{attribute 'c++_compatible'}
FUNCTION_BLOCK UDPConnect IMPLEMENTS ITcIoUdpProtocolRecv
VAR_INPUT
END_VAR
VAR_OUTPUT
END_VAR
VAR
	{attribute 'TcInitSymbol'}
    oid:              OTCID; 
    ipUdp:            ITcIoUdpProtocol;
    updPort:          UINT := 25000;
    nReceivedPakets:  UINT;
    hrInit :          HRESULT;
    hrSend :          HRESULT;
END_VAR

IF ipUdp <> 0 THEN
    ipUdp.CheckReceived();
END_IF

METHOD FB_exit : BOOL
VAR_INPUT
	bInCopyCode : BOOL; // if TRUE, the exit method is called for exiting an instance that is copied afterwards (online change).
END_VAR
IF (NOT bInCopyCode AND ipUdp <> 0) THEN //Shutdown
     ipUdp.UnregisterReceiver(updPort);
    FW_SafeRelease(ADR(ipUdp));
     FB_exit := TRUE;
ELSE
     FB_exit := FALSE;
END_IF
END_METHOD

METHOD FB_init : BOOL
VAR_INPUT
	bInitRetains : BOOL; // if TRUE, the retain variables are initialized (warm start / cold start)
	bInCopyCode : BOOL;  // if TRUE, the instance afterwards gets moved into the copy code (online change)
END_VAR

VAR
    ipSrv: ITComObjectServer;
    hr : HRESULT;
END_VAR
IF NOT bInCopyCode THEN // no online change
    IF ipUdp = 0 THEN
     hrInit := FW_ObjMgr_GetObjectInstance(   oid:=oid, 
    
    iid:=TC_GLOBAL_IID_LIST.IID_ITcIoUdpProtocol, 

    pipUnk:=ADR(ipUdp) );
        IF ( SUCCEEDED(hr) AND ipUdp.RegisterReceiver(updPort, THIS^) = 0 ) THEN //open port
            FB_init := TRUE;
        ELSE
            FB_init := FALSE; 
            FW_SafeRelease(ADR(ipUdp));
        END_IF
    END_IF
END_IF
END_METHOD

METHOD FB_reinit : BOOL
VAR_INPUT
END_VAR
IF (ipUdp <> 0) THEN 
 ipUdp.RegisterReceiver(updPort, THIS^);
END_IF
END_METHOD

{attribute 'object_name' := 'ReceiveData'}
{attribute 'c++_compatible'}
{attribute 'signature_flag' := '33554688'}
{attribute 'pack_mode' := '4'}
{attribute 'show'}
{attribute 'minimal_input_size' := '4'}
METHOD ReceiveData : HRESULT
VAR_INPUT
	ipAddr	: UDINT;
	udpDestPort	: UINT;
	udpSrcPort	: UINT;
	nData	: UDINT;
	pData	: PVOID;
	pVlan	: POINTER TO ETYPE_VLAN_HEADER := 0;
END_VAR

VAR
	i	: ULINT := 0;
END_VAR
nReceivedPakets := nReceivedPakets+1;
//MAIN_UDP.nPaketlaenge := nData;

FOR i := 0 TO 3 DO
	memcpy(ADR(UDP.x[i+1]),pData+((i*3)*8),8);
	memcpy(ADR(UDP.y[i+1]),pData+((i*3+1)*8),8);
	memcpy(ADR(UDP.theta[i+1]),pData+((i*3+2)*8),8);
END_FOR;
END_METHOD

{attribute 'c++_compatible'}
{attribute 'minimal_input_size' := '4'}
{attribute 'pack_mode' := '4'}
{warning 'Methodenimplementierung hinzufügen'}
METHOD TcAddRef : UDINT
END_METHOD

{attribute 'c++_compatible'}
{attribute 'minimal_input_size' := '4'}
{attribute 'pack_mode' := '4'}
{warning 'Methodenimplementierung hinzufügen'}
METHOD TcQueryInterface : HRESULT
VAR_INPUT
	iid	: REFERENCE TO IID;
	pipItf	: POINTER TO PVOID;
END_VAR
END_METHOD

{attribute 'c++_compatible'}
{attribute 'minimal_input_size' := '4'}
{attribute 'pack_mode' := '4'}
{warning 'Methodenimplementierung hinzufügen'}
METHOD TcRelease : UDINT
END_METHOD

END_FUNCTION_BLOCK

(* stored: Version 1.1.0.1, ProductVersion 3.1.4022.3
   POU UDPConnect: Id {f48a780d-9067-4517-b718-1e333e4d91b3}, SpecialFunc None
   Method FB_exit: Id {f8c77def-1015-4a63-9131-8794a85af723}
   Method FB_init: Id {85af01f4-97f3-44d1-bdff-a28ebfe19fb8}
   Method FB_reinit: Id {460b2555-1097-49e1-8a3e-feff2c1020f1}
   Method ReceiveData: Id {df8748c4-1eda-4c5a-9523-38fce868db7a}
   Method TcAddRef: Id {c21f6ce7-d332-4863-a678-81646bd050cb}
   Method TcQueryInterface: Id {d51791d7-5102-4fa7-8dd6-fb98a6db8305}
   Method TcRelease: Id {12802f4d-9a9d-4391-b560-1f25bff2d2cb} *)
